// TIA Portal V20 export
TYPE "LER_TypeFATMode_HoursTest"
// stored: Access Published
   STRUCT
      ProcessValue : "LER_TypeFATMode_HoursTest_ProcessValue";
      SetValue { S7_SetPoint := 'True'} : "LER_TypeFATMode_HoursTest_SetValue";
   END_STRUCT;
END_TYPE
